SUBAPPLICATION Uebung_006c_AX (* SR-Flip-Flop mit IB auf DI_REPEAT *)
  (* Standard: 61499-2; Description: Copyright (c) 2023 Meisterschulen am Ostbahnhof This program and the accompanying materials are made available under the terms of the Eclipse Public License 2.0 which is available at https://www.eclipse.org/legal/epl-2.0/ SPDX-License-Identifier: EPL-2.0 *)
  (* Version 1.0, 2023-10-23, Franz Höpfinger, Meisterschulen am Ostbahnhof, initial API and implementation and/or initial documentation *)
  PACKAGE Uebungen;
  IMPORT logiBUS::io::DI::logiBUS_DI::Input_I1;
  IMPORT logiBUS::io::DI::logiBUS_DI::Input_I2;
  IMPORT logiBUS::io::DI::logiBUS_DI_Events::BUTTON_PRESS_REPEAT;
  IMPORT logiBUS::io::DQ::logiBUS_DO::Output_Q1;
  IMPORT logiBUS::io::DQ::logiBUS_DO::Output_Q2;
  IMPORT logiBUS::io::DQ::logiBUS_DO::Output_Q3;
  IMPORT logiBUS::io::DQ::logiBUS_DO::Output_Q4;
  IMPORT logiBUS::io::DQ::logiBUS_DO::Output_Q5;
  IMPORT logiBUS::io::DQ::logiBUS_DO::Output_Q6;
  IMPORT logiBUS::io::DQ::logiBUS_DO::Output_Q7;
  IMPORT logiBUS::io::DQ::logiBUS_DO::Output_Q8;
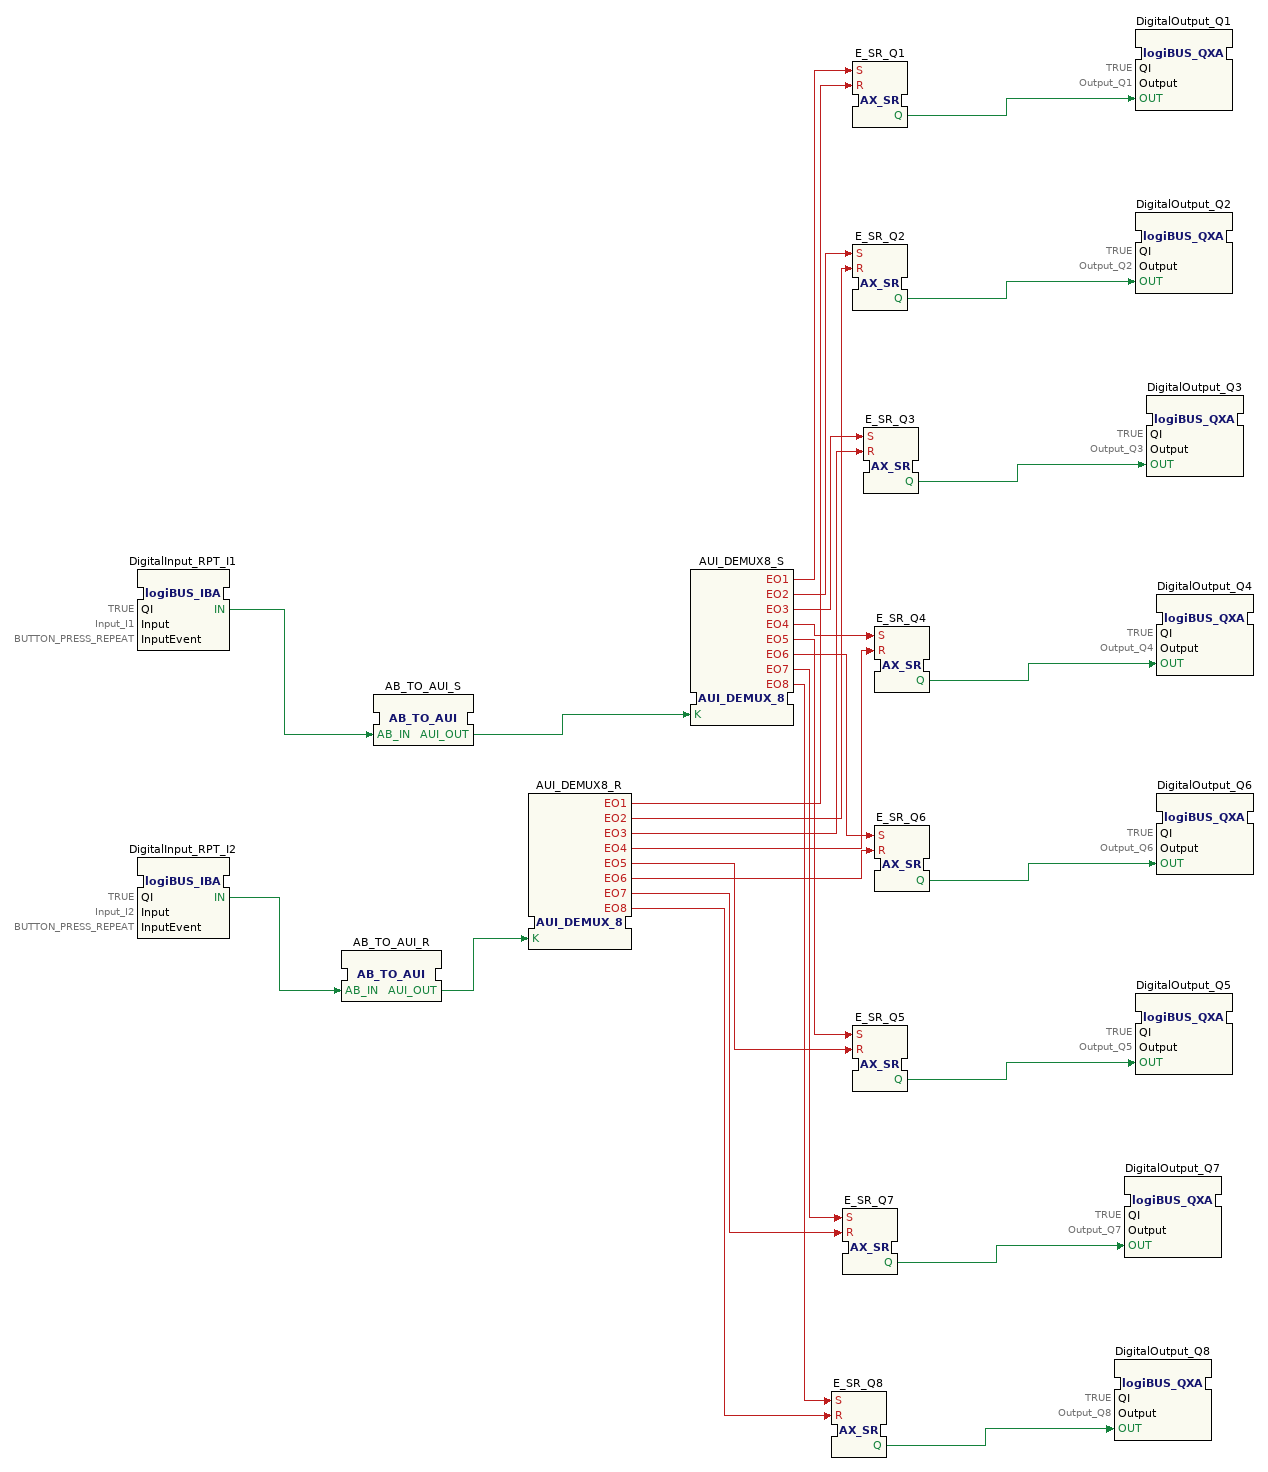
  FBS
    DigitalOutput_Q1 : logiBUS::io::DQ::logiBUS_QXA(QI := TRUE, Output := Output_Q1);
    DigitalInput_RPT_I1 : logiBUS::io::DI::logiBUS_IBA(QI := TRUE, Input := Input_I1, InputEvent := BUTTON_PRESS_REPEAT);
    DigitalInput_RPT_I2 : logiBUS::io::DI::logiBUS_IBA(QI := TRUE, Input := Input_I2, InputEvent := BUTTON_PRESS_REPEAT);
    E_SR_Q1 : adapter::events::unidirectional::AX_SR;
    E_SR_Q2 : adapter::events::unidirectional::AX_SR;
    DigitalOutput_Q2 : logiBUS::io::DQ::logiBUS_QXA(QI := TRUE, Output := Output_Q2);
    DigitalOutput_Q3 : logiBUS::io::DQ::logiBUS_QXA(QI := TRUE, Output := Output_Q3);
    DigitalOutput_Q4 : logiBUS::io::DQ::logiBUS_QXA(QI := TRUE, Output := Output_Q4);
    E_SR_Q5 : adapter::events::unidirectional::AX_SR;
    E_SR_Q6 : adapter::events::unidirectional::AX_SR;
    DigitalOutput_Q5 : logiBUS::io::DQ::logiBUS_QXA(QI := TRUE, Output := Output_Q5);
    DigitalOutput_Q6 : logiBUS::io::DQ::logiBUS_QXA(QI := TRUE, Output := Output_Q6);
    DigitalOutput_Q7 : logiBUS::io::DQ::logiBUS_QXA(QI := TRUE, Output := Output_Q7);
    DigitalOutput_Q8 : logiBUS::io::DQ::logiBUS_QXA(QI := TRUE, Output := Output_Q8);
    AUI_DEMUX8_S : adapter::events::unidirectional::AUI_DEMUX_8;
    AUI_DEMUX8_R : adapter::events::unidirectional::AUI_DEMUX_8;
    E_SR_Q3 : adapter::events::unidirectional::AX_SR;
    E_SR_Q4 : adapter::events::unidirectional::AX_SR;
    E_SR_Q7 : adapter::events::unidirectional::AX_SR;
    E_SR_Q8 : adapter::events::unidirectional::AX_SR;
    AB_TO_AUI_S : adapter::conversion::unidirectional::AB_TO_AUI;
    AB_TO_AUI_R : adapter::conversion::unidirectional::AB_TO_AUI;
  END_FBS
  EVENT_CONNECTIONS
    AUI_DEMUX8_S.EO1 TO E_SR_Q1.S;
    AUI_DEMUX8_S.EO2 TO E_SR_Q2.S;
    AUI_DEMUX8_S.EO3 TO E_SR_Q3.S;
    AUI_DEMUX8_S.EO4 TO E_SR_Q4.S;
    AUI_DEMUX8_S.EO5 TO E_SR_Q5.S;
    AUI_DEMUX8_S.EO6 TO E_SR_Q6.S;
    AUI_DEMUX8_S.EO7 TO E_SR_Q7.S;
    AUI_DEMUX8_S.EO8 TO E_SR_Q8.S;
    AUI_DEMUX8_R.EO1 TO E_SR_Q1.R;
    AUI_DEMUX8_R.EO2 TO E_SR_Q2.R;
    AUI_DEMUX8_R.EO3 TO E_SR_Q3.R;
    AUI_DEMUX8_R.EO4 TO E_SR_Q4.R;
    AUI_DEMUX8_R.EO5 TO E_SR_Q5.R;
    AUI_DEMUX8_R.EO6 TO E_SR_Q6.R;
    AUI_DEMUX8_R.EO7 TO E_SR_Q7.R;
    AUI_DEMUX8_R.EO8 TO E_SR_Q8.R;
  END_CONNECTIONS
  ADAPTER_CONNECTIONS
    DigitalInput_RPT_I1.IN TO AB_TO_AUI_S.AB_IN;
    AB_TO_AUI_S.AUI_OUT TO AUI_DEMUX8_S.K;
    DigitalInput_RPT_I2.IN TO AB_TO_AUI_R.AB_IN;
    AB_TO_AUI_R.AUI_OUT TO AUI_DEMUX8_R.K;
    E_SR_Q1.Q TO DigitalOutput_Q1.OUT;
    E_SR_Q2.Q TO DigitalOutput_Q2.OUT;
    E_SR_Q3.Q TO DigitalOutput_Q3.OUT;
    E_SR_Q4.Q TO DigitalOutput_Q4.OUT;
    E_SR_Q5.Q TO DigitalOutput_Q5.OUT;
    E_SR_Q6.Q TO DigitalOutput_Q6.OUT;
    E_SR_Q7.Q TO DigitalOutput_Q7.OUT;
    E_SR_Q8.Q TO DigitalOutput_Q8.OUT;
  END_CONNECTIONS
END_SUBAPPLICATION
